TYPE ExampleDomain_Io :
STRUCT
	in			: ExampleDomain_Io_In;
	out			: ExampleDomain_Io_Out;
END_STRUCT
END_TYPE

(* stored: Version 1.1.0.1
   DUT ExampleDomain_Io: Id {35b6a7b8-d5da-4e7e-a8f9-6d81a6ab5f98} *)
